TYPE Mat37 : ARRAY[1..3, 1..7] OF LREAL; END_TYPE

(* stored: Version 1.1.0.1, ProductVersion 3.1.4024.12
   DUT Mat37: Id {1604c40f-b191-40be-a318-dd99118ec86b} *)
